Staubli VAL3: pp.dtx

bool bBool1 = true
jointRx jHome
mdesc mNomSpeed
mdesc mSlow = {accel=25, vel=25, decel=25, tmax=25, rmax=25}
num nRep
pointRx pPointrx1[3]
  [0] = {x=611.54, y=-334.812005, z=260.499354, rx=-4.959689, ry=154.036634, rz=-5.509255, fatherId=world[0]}
  [1] = {x=739.655424, y=-22.141465, z=103.226279, rx=9.330921, ry=168.093288, rz=-33.667519, fatherId=world[0]}
  [2] = {x=330.134697, y=799.531714, z=-139.574889, rx=170.585193, ry=-7.909797, rz=71.354806, fatherId=world[0]}
tool tTool1 = {fatherId=flange[0], ioLink=valve1}
screen Interfaz
num nPact[2]
num nPdes[2]
bool bBool2 = true
